// The verifier's task entry point.
//
// The floor check stands alone and runs first: it proves the harness can run a
// test at all, WITHOUT using the harness to prove it. Read PRG_FloorCheck.AllGood
// before trusting anything in PRG_UnitTests - if the runner is broken, every test
// reports NotStarted and that looks exactly like a wiring mistake.
PROGRAM MAIN

PRG_FloorCheck();
PRG_UnitTests();

END_PROGRAM

(* stored: Version 1.1.0.1, ProductVersion 3.1.4026.18
   POU MAIN: Id {6ad23a12-ff60-4084-95d3-efc5edf615eb}, SpecialFunc None *)
